VAR_GLOBAL CONSTANT
	ALARM_INVALID_CONTEXT_ID	: DINT := 0;
	ALARM_INVALID_INDEX			: DINT := -1;
	ALARM_ARG_STACK_SIZE		: DINT := 255;
	ALARM_TEXT_SIZE				: INT := 255;
END_VAR

(* stored: Version 1.1.0.1, ProductVersion 3.1.4024.15
   GVL GVL_Alarms: Id {2c67669b-06d4-439a-b056-792cfc801adc} *)
